// TIA Portal V19 export
TYPE "LEXCHANGETRAY_typeLogistics_recieve_interface"
// stored: Access Published
   STRUCT
      roller : "LEXCHANGETRAY_typeLogistics_toRollerRecieve";
   END_STRUCT;
END_TYPE
